KUKA KRL data list: D15_DCD_PICK.dat

&ACCESS RVO
&REL 1
&PARAM DISKPATH = KRC:\R1\Program\SbtComm001Main\D
DEFDAT D15_DCD_PICK
;FOLD EXTERNAL DECLARATIONS;%{PE}%MKUKATPBASIS,%CEXT,%VCOMMON,%P
;FOLD BASISTECH EXT;%{PE}%MKUKATPBASIS,%CEXT,%VEXT,%P
EXT  BAS (BAS_COMMAND  :IN,REAL  :IN )
DECL INT SUCCESS
DECL int key
DECL int DicisionCode
DECL STATE_T State
DECL INT Offset
CHAR Msg[256]
;ENDFOLD (BASISTECH EXT)
;FOLD USER EXT;%{E}%MKUKATPUSER,%CEXT,%VEXT,%P
;Make your modifications here

;ENDFOLD (USER EXT)
;ENDFOLD (EXTERNAL DECLARATIONS)
ENDDAT
